TYPE (* ISO Part 5 name field structure according to IFM conventions *)
  (* Version 1.0, 2025-09-04, Coding-Assistent *)
  ISONAMEFIELD_T : STRUCT
    bSelfConf : BOOL; (* Self-configurable-address ECU? *)
    bIndGroup : BYTE; (* NAMES associated with industries (0..7, 255 = Filter for all) *)
    bDevClassInst : BYTE; (* Identifier if a device class more than 1 times in net (0..15, 255 = Filter for all) *)
    bDevClass : BYTE; (* ISO Defined (0..127, 255 = Filter for all) *)
    bReserved : BOOL; (* Reserved (not used) *)
    bFunction : WORD; (* ISO defined, -> SA (0..255, 65535 = Filter for all) *)
    bFunctionInst : BYTE; (* Subgroup of function (0..31, 255 = Filter for all) *)
    bEcuInstance : BYTE; (* Which ECU associated with a given function (0..7, 255 = Filter for all) *)
    wManufCode : WORD; (* ISO defined (0..2047, 65535 = Filter for all) *)
    dwIdentNumb : DWORD; (* Used when the NAME is not unique in same network (0..2047, 4294967295 = Filter for all) *)
  END_STRUCT;
END_TYPE
